Staubli VAL3: exeWZone.pgx

program exeWzone(tool x_tTool, point x_pPoint, frame x_fFrame, num x_Dx, num x_Dy, num x_Dz, dio x_dOut)
  local bool l_bXok
  local bool l_bYok
  local bool l_bZok
  local point l_pHere
begin
  while true
    l_pHere=here(x_tTool,x_fFrame)
    l_bXok=l_pHere.trsf.x>x_pPoint.trsf.x-x_Dx/2 and l_pHere.trsf.x<x_pPoint.trsf.x+x_Dx/2
    l_bYok=l_pHere.trsf.y>x_pPoint.trsf.y-x_Dy/2 and l_pHere.trsf.y<x_pPoint.trsf.y+x_Dy/2
    l_bZok=l_pHere.trsf.z>x_pPoint.trsf.z-x_Dz/2 and l_pHere.trsf.z<x_pPoint.trsf.z+x_Dz/2
    if l_bXok and l_bYok and l_bZok
      x_dOut=false
    else
      x_dOut=true
    endIf
    delay(0)
  endWhile
end
